PROGRAM Config_Slow
VAR
	
	
	Once				:BOOL :=TRUE;
	saving_config		:BOOL :=FALSE;		
END_VAR

IF Clock.DateTimeInitialised THEN
   	//Config_Counter:=Config_Counter+1;
	//config_count:=config_count+1;
	//IF config_count = 30 THEN
	//	Config();
	//	config_count:=0;
	//END_IF
	IF Config.Initialised() = FALSE THEN
		Config();
	ELSIF Once = TRUE THEN
		Message := 'Data Loaded';
		Once := FALSE;
	END_IF
	
	
	IF Config_Request = TRUE AND saving_config = FALSE THEN
		Config_Request:=FALSE;
		saving_config:=TRUE;
		config_count:=0;

	END_IF
	
	IF saving_config AND config_count <=2500 THEN
		Config();
		config_count:=config_count+1;
	END_IF
	
	IF config_count = 2500 THEN
		saving_config:= FALSE;
		config_count :=0;
		IF config_request = FALSE THEN
			Message := 'Operation Configured';
		END_IF
	END_IF	

END_IF

END_PROGRAM

(* stored: Version 1.1.0.1, ProductVersion 3.1.4020.12
   POU Config_Slow: Id {68820ce0-f190-48fe-919d-63c0e6e8e6eb}, SpecialFunc None *)
